PROGRAM TempCtrl
VAR

END_VAR

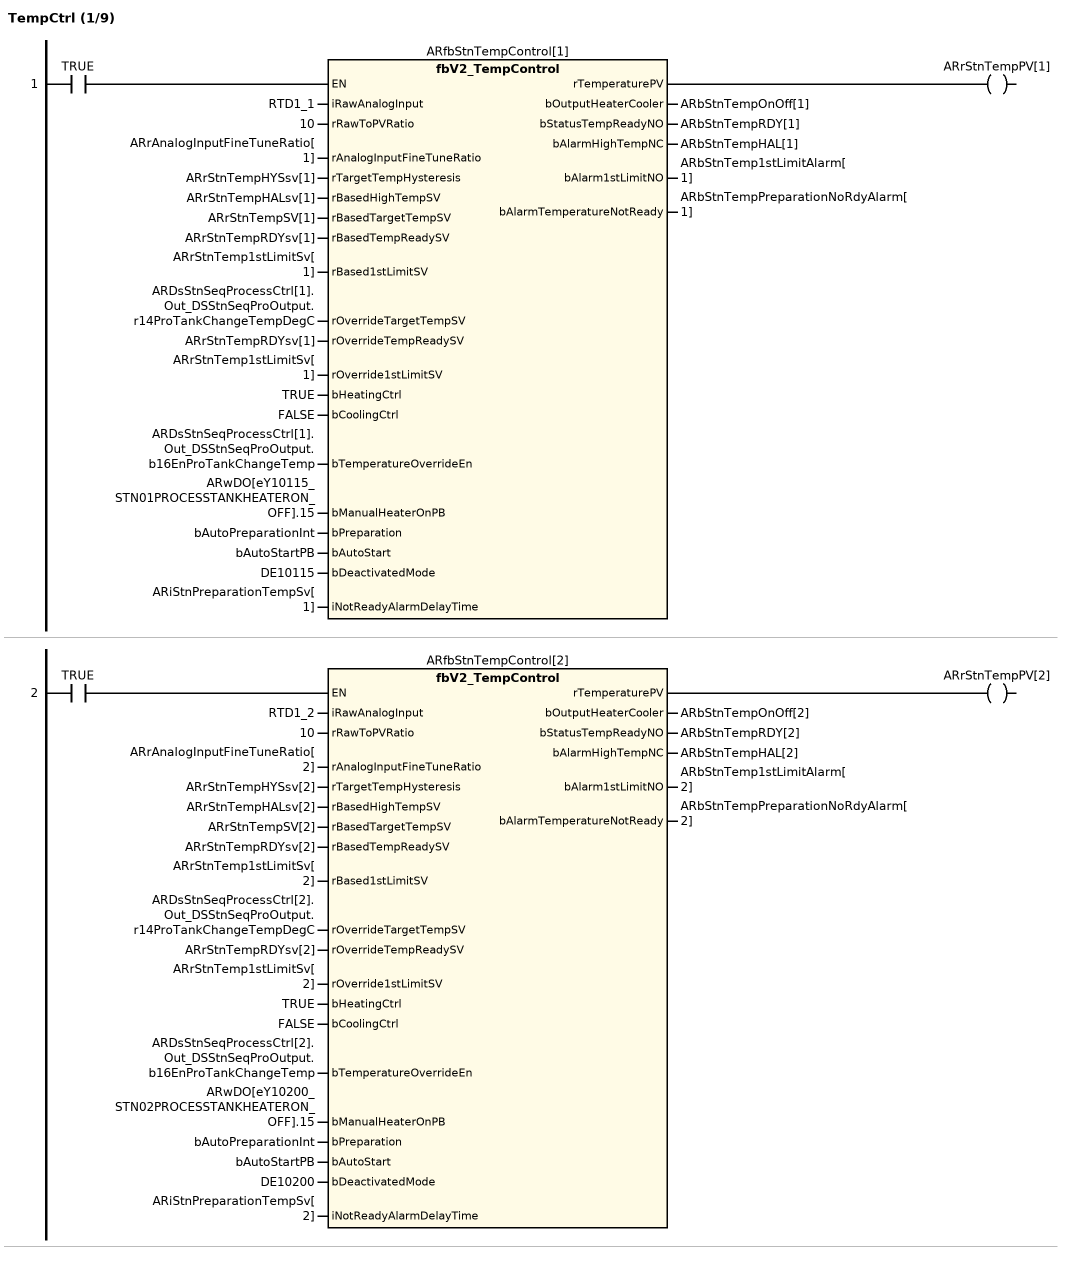
// NETWORK 1
ARfbStnTempControl[1](
    iRawAnalogInput := RTD1_1,
    rRawToPVRatio := 10,
    rAnalogInputFineTuneRatio := ARrAnalogInputFineTuneRatio[1],
    rTargetTempHysteresis := ARrStnTempHYSsv[1],
    rBasedHighTempSV := ARrStnTempHALsv[1],
    rBasedTargetTempSV := ARrStnTempSV[1],
    rBasedTempReadySV := ARrStnTempRDYsv[1],
    rBased1stLimitSV := ARrStnTemp1stLimitSv[1],
    rOverrideTargetTempSV := ARDsStnSeqProcessCtrl[1].Out_DSStnSeqProOutput.r14ProTankChangeTempDegC,
    rOverrideTempReadySV := ARrStnTempRDYsv[1],
    rOverride1stLimitSV := ARrStnTemp1stLimitSv[1],
    bHeatingCtrl := TRUE,
    bCoolingCtrl := FALSE,
    bTemperatureOverrideEn := ARDsStnSeqProcessCtrl[1].Out_DSStnSeqProOutput.b16EnProTankChangeTemp,
    bManualHeaterOnPB := ARwDO[eY10115_STN01PROCESSTANKHEATERON_OFF].15,
    bPreparation := bAutoPreparationInt,
    bAutoStart := bAutoStartPB,
    bDeactivatedMode := DE10115,
    iNotReadyAlarmDelayTime := ARiStnPreparationTempSv[1],
    bOutputHeaterCooler => ARbStnTempOnOff[1],
    bStatusTempReadyNO => ARbStnTempRDY[1],
    bAlarmHighTempNC => ARbStnTempHAL[1],
    bAlarm1stLimitNO => ARbStnTemp1stLimitAlarm[1],
    bAlarmTemperatureNotReady => ARbStnTempPreparationNoRdyAlarm[1]); // fbV2_TempControl
ARrStnTempPV[1] := ARfbStnTempControl[1].rTemperaturePV;

// NETWORK 2
ARfbStnTempControl[2](
    iRawAnalogInput := RTD1_2,
    rRawToPVRatio := 10,
    rAnalogInputFineTuneRatio := ARrAnalogInputFineTuneRatio[2],
    rTargetTempHysteresis := ARrStnTempHYSsv[2],
    rBasedHighTempSV := ARrStnTempHALsv[2],
    rBasedTargetTempSV := ARrStnTempSV[2],
    rBasedTempReadySV := ARrStnTempRDYsv[2],
    rBased1stLimitSV := ARrStnTemp1stLimitSv[2],
    rOverrideTargetTempSV := ARDsStnSeqProcessCtrl[2].Out_DSStnSeqProOutput.r14ProTankChangeTempDegC,
    rOverrideTempReadySV := ARrStnTempRDYsv[2],
    rOverride1stLimitSV := ARrStnTemp1stLimitSv[2],
    bHeatingCtrl := TRUE,
    bCoolingCtrl := FALSE,
    bTemperatureOverrideEn := ARDsStnSeqProcessCtrl[2].Out_DSStnSeqProOutput.b16EnProTankChangeTemp,
    bManualHeaterOnPB := ARwDO[eY10200_STN02PROCESSTANKHEATERON_OFF].15,
    bPreparation := bAutoPreparationInt,
    bAutoStart := bAutoStartPB,
    bDeactivatedMode := DE10200,
    iNotReadyAlarmDelayTime := ARiStnPreparationTempSv[2],
    bOutputHeaterCooler => ARbStnTempOnOff[2],
    bStatusTempReadyNO => ARbStnTempRDY[2],
    bAlarmHighTempNC => ARbStnTempHAL[2],
    bAlarm1stLimitNO => ARbStnTemp1stLimitAlarm[2],
    bAlarmTemperatureNotReady => ARbStnTempPreparationNoRdyAlarm[2]); // fbV2_TempControl
ARrStnTempPV[2] := ARfbStnTempControl[2].rTemperaturePV;

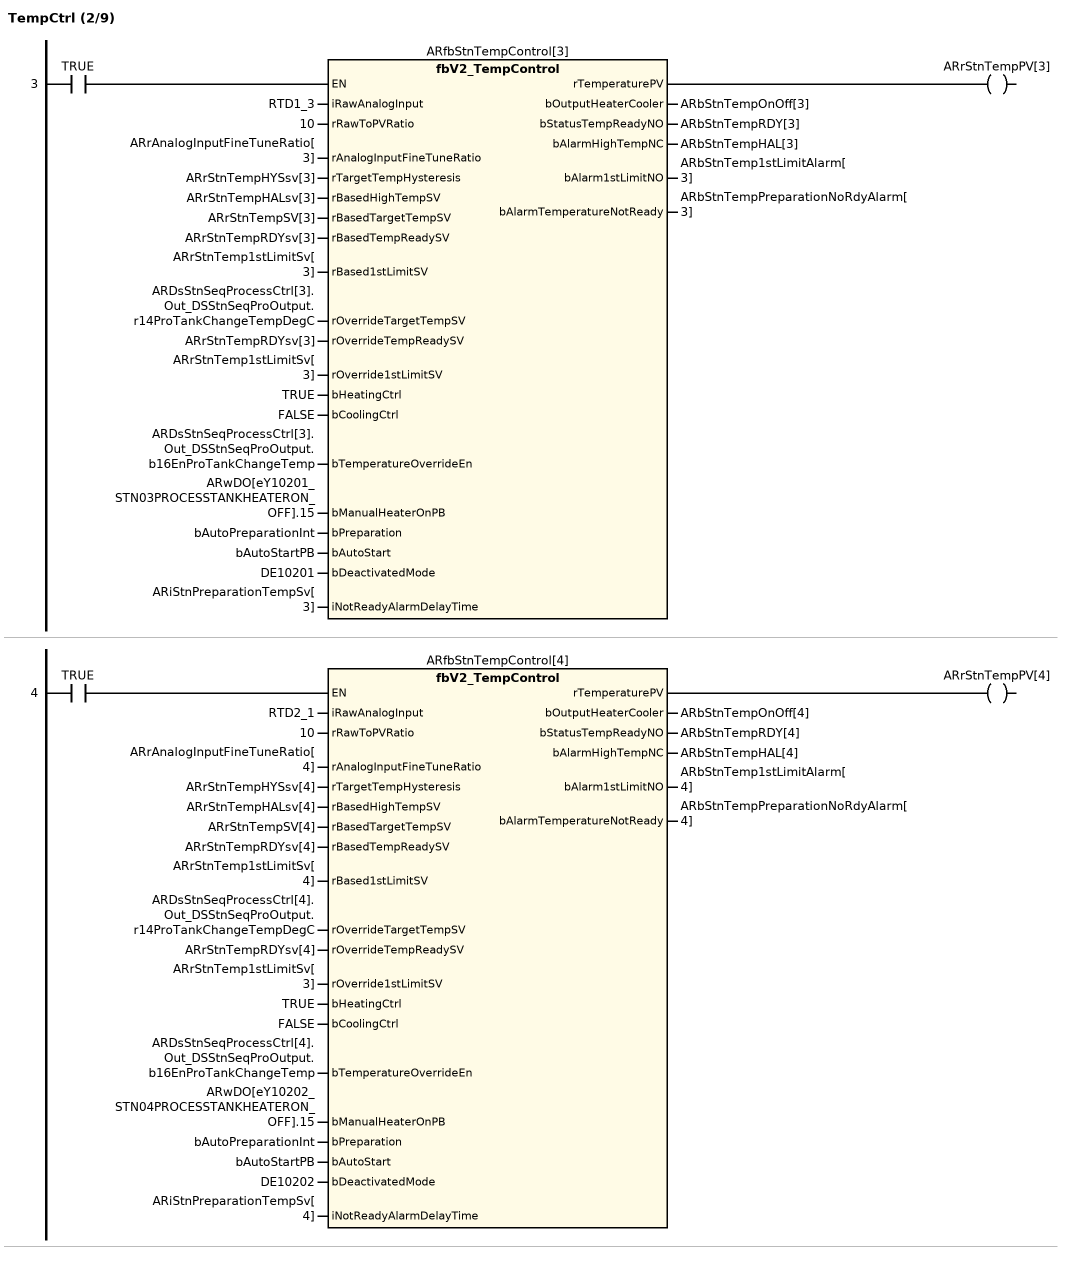
// NETWORK 3
ARfbStnTempControl[3](
    iRawAnalogInput := RTD1_3,
    rRawToPVRatio := 10,
    rAnalogInputFineTuneRatio := ARrAnalogInputFineTuneRatio[3],
    rTargetTempHysteresis := ARrStnTempHYSsv[3],
    rBasedHighTempSV := ARrStnTempHALsv[3],
    rBasedTargetTempSV := ARrStnTempSV[3],
    rBasedTempReadySV := ARrStnTempRDYsv[3],
    rBased1stLimitSV := ARrStnTemp1stLimitSv[3],
    rOverrideTargetTempSV := ARDsStnSeqProcessCtrl[3].Out_DSStnSeqProOutput.r14ProTankChangeTempDegC,
    rOverrideTempReadySV := ARrStnTempRDYsv[3],
    rOverride1stLimitSV := ARrStnTemp1stLimitSv[3],
    bHeatingCtrl := TRUE,
    bCoolingCtrl := FALSE,
    bTemperatureOverrideEn := ARDsStnSeqProcessCtrl[3].Out_DSStnSeqProOutput.b16EnProTankChangeTemp,
    bManualHeaterOnPB := ARwDO[eY10201_STN03PROCESSTANKHEATERON_OFF].15,
    bPreparation := bAutoPreparationInt,
    bAutoStart := bAutoStartPB,
    bDeactivatedMode := DE10201,
    iNotReadyAlarmDelayTime := ARiStnPreparationTempSv[3],
    bOutputHeaterCooler => ARbStnTempOnOff[3],
    bStatusTempReadyNO => ARbStnTempRDY[3],
    bAlarmHighTempNC => ARbStnTempHAL[3],
    bAlarm1stLimitNO => ARbStnTemp1stLimitAlarm[3],
    bAlarmTemperatureNotReady => ARbStnTempPreparationNoRdyAlarm[3]); // fbV2_TempControl
ARrStnTempPV[3] := ARfbStnTempControl[3].rTemperaturePV;

// NETWORK 4
ARfbStnTempControl[4](
    iRawAnalogInput := RTD2_1,
    rRawToPVRatio := 10,
    rAnalogInputFineTuneRatio := ARrAnalogInputFineTuneRatio[4],
    rTargetTempHysteresis := ARrStnTempHYSsv[4],
    rBasedHighTempSV := ARrStnTempHALsv[4],
    rBasedTargetTempSV := ARrStnTempSV[4],
    rBasedTempReadySV := ARrStnTempRDYsv[4],
    rBased1stLimitSV := ARrStnTemp1stLimitSv[4],
    rOverrideTargetTempSV := ARDsStnSeqProcessCtrl[4].Out_DSStnSeqProOutput.r14ProTankChangeTempDegC,
    rOverrideTempReadySV := ARrStnTempRDYsv[4],
    rOverride1stLimitSV := ARrStnTemp1stLimitSv[3],
    bHeatingCtrl := TRUE,
    bCoolingCtrl := FALSE,
    bTemperatureOverrideEn := ARDsStnSeqProcessCtrl[4].Out_DSStnSeqProOutput.b16EnProTankChangeTemp,
    bManualHeaterOnPB := ARwDO[eY10202_STN04PROCESSTANKHEATERON_OFF].15,
    bPreparation := bAutoPreparationInt,
    bAutoStart := bAutoStartPB,
    bDeactivatedMode := DE10202,
    iNotReadyAlarmDelayTime := ARiStnPreparationTempSv[4],
    bOutputHeaterCooler => ARbStnTempOnOff[4],
    bStatusTempReadyNO => ARbStnTempRDY[4],
    bAlarmHighTempNC => ARbStnTempHAL[4],
    bAlarm1stLimitNO => ARbStnTemp1stLimitAlarm[4],
    bAlarmTemperatureNotReady => ARbStnTempPreparationNoRdyAlarm[4]); // fbV2_TempControl
ARrStnTempPV[4] := ARfbStnTempControl[4].rTemperaturePV;

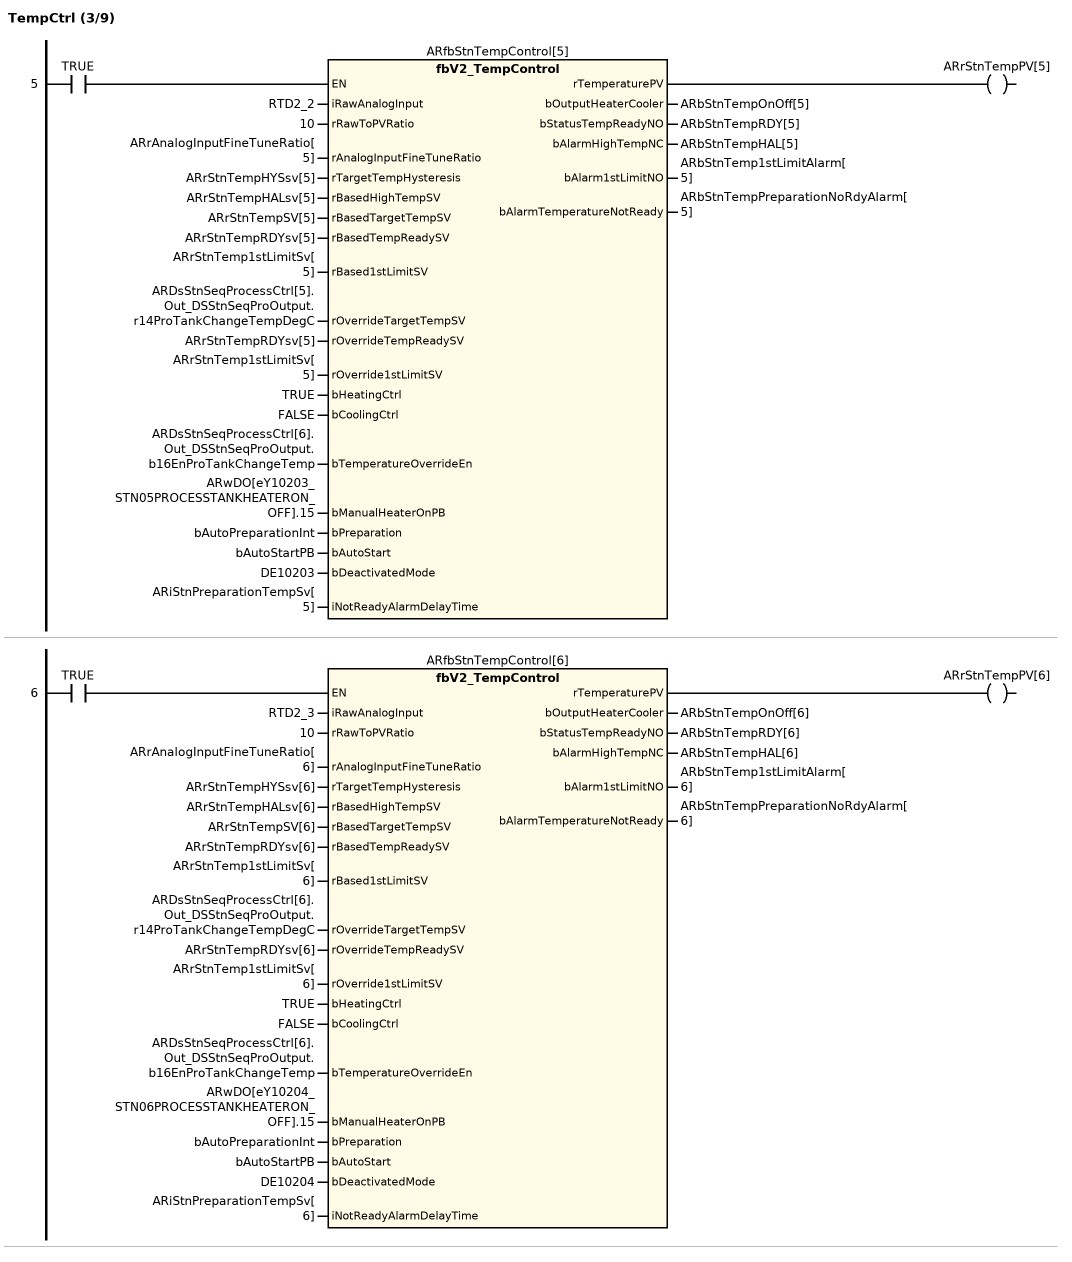
// NETWORK 5
ARfbStnTempControl[5](
    iRawAnalogInput := RTD2_2,
    rRawToPVRatio := 10,
    rAnalogInputFineTuneRatio := ARrAnalogInputFineTuneRatio[5],
    rTargetTempHysteresis := ARrStnTempHYSsv[5],
    rBasedHighTempSV := ARrStnTempHALsv[5],
    rBasedTargetTempSV := ARrStnTempSV[5],
    rBasedTempReadySV := ARrStnTempRDYsv[5],
    rBased1stLimitSV := ARrStnTemp1stLimitSv[5],
    rOverrideTargetTempSV := ARDsStnSeqProcessCtrl[5].Out_DSStnSeqProOutput.r14ProTankChangeTempDegC,
    rOverrideTempReadySV := ARrStnTempRDYsv[5],
    rOverride1stLimitSV := ARrStnTemp1stLimitSv[5],
    bHeatingCtrl := TRUE,
    bCoolingCtrl := FALSE,
    bTemperatureOverrideEn := ARDsStnSeqProcessCtrl[6].Out_DSStnSeqProOutput.b16EnProTankChangeTemp,
    bManualHeaterOnPB := ARwDO[eY10203_STN05PROCESSTANKHEATERON_OFF].15,
    bPreparation := bAutoPreparationInt,
    bAutoStart := bAutoStartPB,
    bDeactivatedMode := DE10203,
    iNotReadyAlarmDelayTime := ARiStnPreparationTempSv[5],
    bOutputHeaterCooler => ARbStnTempOnOff[5],
    bStatusTempReadyNO => ARbStnTempRDY[5],
    bAlarmHighTempNC => ARbStnTempHAL[5],
    bAlarm1stLimitNO => ARbStnTemp1stLimitAlarm[5],
    bAlarmTemperatureNotReady => ARbStnTempPreparationNoRdyAlarm[5]); // fbV2_TempControl
ARrStnTempPV[5] := ARfbStnTempControl[5].rTemperaturePV;

// NETWORK 6
ARfbStnTempControl[6](
    iRawAnalogInput := RTD2_3,
    rRawToPVRatio := 10,
    rAnalogInputFineTuneRatio := ARrAnalogInputFineTuneRatio[6],
    rTargetTempHysteresis := ARrStnTempHYSsv[6],
    rBasedHighTempSV := ARrStnTempHALsv[6],
    rBasedTargetTempSV := ARrStnTempSV[6],
    rBasedTempReadySV := ARrStnTempRDYsv[6],
    rBased1stLimitSV := ARrStnTemp1stLimitSv[6],
    rOverrideTargetTempSV := ARDsStnSeqProcessCtrl[6].Out_DSStnSeqProOutput.r14ProTankChangeTempDegC,
    rOverrideTempReadySV := ARrStnTempRDYsv[6],
    rOverride1stLimitSV := ARrStnTemp1stLimitSv[6],
    bHeatingCtrl := TRUE,
    bCoolingCtrl := FALSE,
    bTemperatureOverrideEn := ARDsStnSeqProcessCtrl[6].Out_DSStnSeqProOutput.b16EnProTankChangeTemp,
    bManualHeaterOnPB := ARwDO[eY10204_STN06PROCESSTANKHEATERON_OFF].15,
    bPreparation := bAutoPreparationInt,
    bAutoStart := bAutoStartPB,
    bDeactivatedMode := DE10204,
    iNotReadyAlarmDelayTime := ARiStnPreparationTempSv[6],
    bOutputHeaterCooler => ARbStnTempOnOff[6],
    bStatusTempReadyNO => ARbStnTempRDY[6],
    bAlarmHighTempNC => ARbStnTempHAL[6],
    bAlarm1stLimitNO => ARbStnTemp1stLimitAlarm[6],
    bAlarmTemperatureNotReady => ARbStnTempPreparationNoRdyAlarm[6]); // fbV2_TempControl
ARrStnTempPV[6] := ARfbStnTempControl[6].rTemperaturePV;

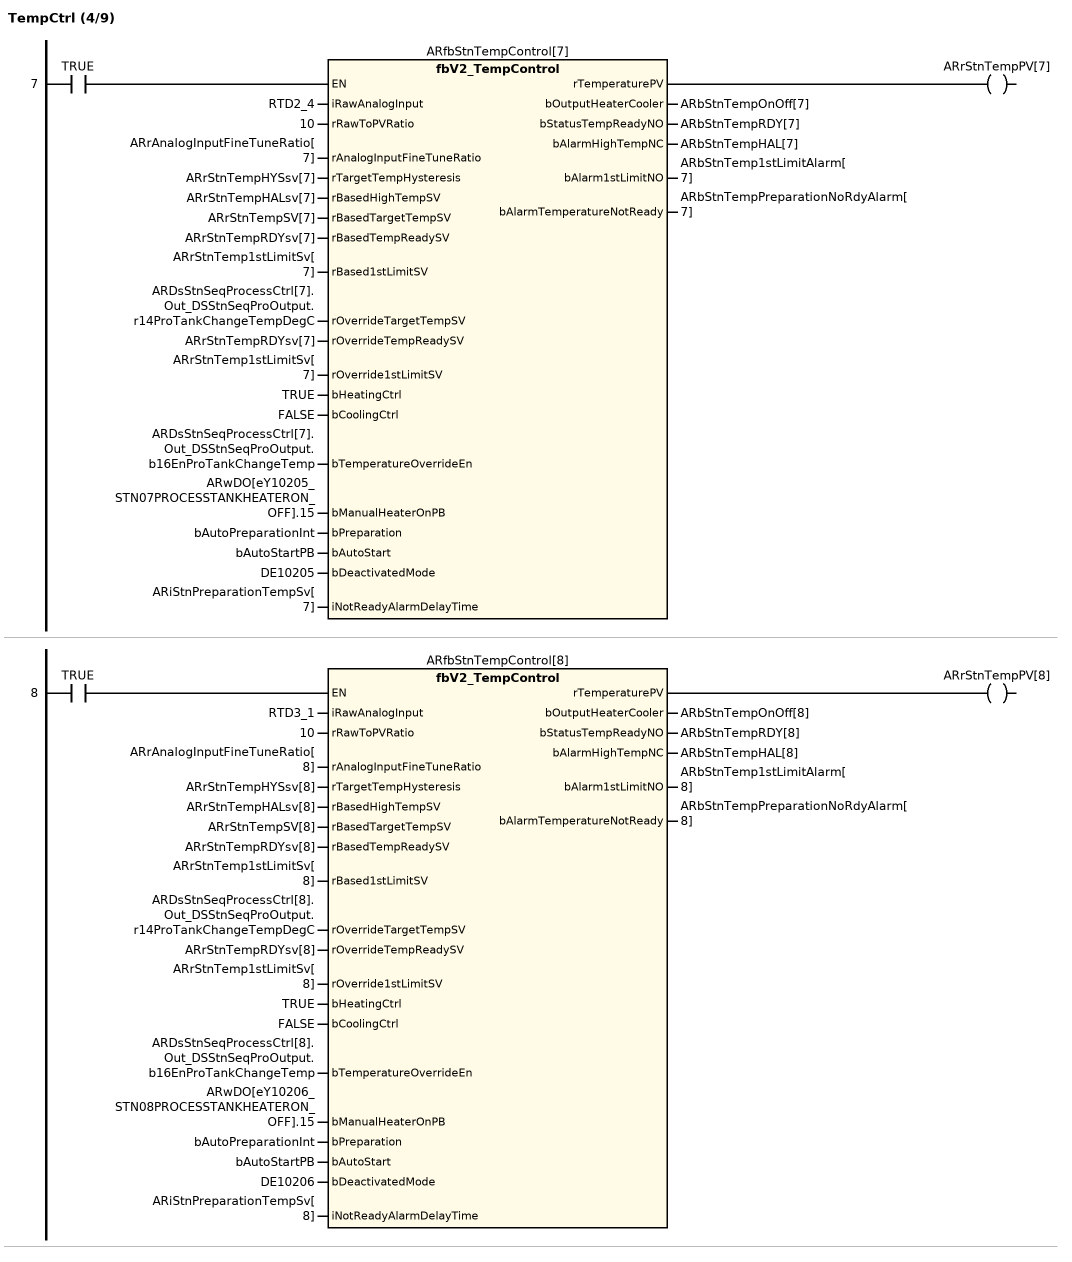
// NETWORK 7
ARfbStnTempControl[7](
    iRawAnalogInput := RTD2_4,
    rRawToPVRatio := 10,
    rAnalogInputFineTuneRatio := ARrAnalogInputFineTuneRatio[7],
    rTargetTempHysteresis := ARrStnTempHYSsv[7],
    rBasedHighTempSV := ARrStnTempHALsv[7],
    rBasedTargetTempSV := ARrStnTempSV[7],
    rBasedTempReadySV := ARrStnTempRDYsv[7],
    rBased1stLimitSV := ARrStnTemp1stLimitSv[7],
    rOverrideTargetTempSV := ARDsStnSeqProcessCtrl[7].Out_DSStnSeqProOutput.r14ProTankChangeTempDegC,
    rOverrideTempReadySV := ARrStnTempRDYsv[7],
    rOverride1stLimitSV := ARrStnTemp1stLimitSv[7],
    bHeatingCtrl := TRUE,
    bCoolingCtrl := FALSE,
    bTemperatureOverrideEn := ARDsStnSeqProcessCtrl[7].Out_DSStnSeqProOutput.b16EnProTankChangeTemp,
    bManualHeaterOnPB := ARwDO[eY10205_STN07PROCESSTANKHEATERON_OFF].15,
    bPreparation := bAutoPreparationInt,
    bAutoStart := bAutoStartPB,
    bDeactivatedMode := DE10205,
    iNotReadyAlarmDelayTime := ARiStnPreparationTempSv[7],
    bOutputHeaterCooler => ARbStnTempOnOff[7],
    bStatusTempReadyNO => ARbStnTempRDY[7],
    bAlarmHighTempNC => ARbStnTempHAL[7],
    bAlarm1stLimitNO => ARbStnTemp1stLimitAlarm[7],
    bAlarmTemperatureNotReady => ARbStnTempPreparationNoRdyAlarm[7]); // fbV2_TempControl
ARrStnTempPV[7] := ARfbStnTempControl[7].rTemperaturePV;

// NETWORK 8
ARfbStnTempControl[8](
    iRawAnalogInput := RTD3_1,
    rRawToPVRatio := 10,
    rAnalogInputFineTuneRatio := ARrAnalogInputFineTuneRatio[8],
    rTargetTempHysteresis := ARrStnTempHYSsv[8],
    rBasedHighTempSV := ARrStnTempHALsv[8],
    rBasedTargetTempSV := ARrStnTempSV[8],
    rBasedTempReadySV := ARrStnTempRDYsv[8],
    rBased1stLimitSV := ARrStnTemp1stLimitSv[8],
    rOverrideTargetTempSV := ARDsStnSeqProcessCtrl[8].Out_DSStnSeqProOutput.r14ProTankChangeTempDegC,
    rOverrideTempReadySV := ARrStnTempRDYsv[8],
    rOverride1stLimitSV := ARrStnTemp1stLimitSv[8],
    bHeatingCtrl := TRUE,
    bCoolingCtrl := FALSE,
    bTemperatureOverrideEn := ARDsStnSeqProcessCtrl[8].Out_DSStnSeqProOutput.b16EnProTankChangeTemp,
    bManualHeaterOnPB := ARwDO[eY10206_STN08PROCESSTANKHEATERON_OFF].15,
    bPreparation := bAutoPreparationInt,
    bAutoStart := bAutoStartPB,
    bDeactivatedMode := DE10206,
    iNotReadyAlarmDelayTime := ARiStnPreparationTempSv[8],
    bOutputHeaterCooler => ARbStnTempOnOff[8],
    bStatusTempReadyNO => ARbStnTempRDY[8],
    bAlarmHighTempNC => ARbStnTempHAL[8],
    bAlarm1stLimitNO => ARbStnTemp1stLimitAlarm[8],
    bAlarmTemperatureNotReady => ARbStnTempPreparationNoRdyAlarm[8]); // fbV2_TempControl
ARrStnTempPV[8] := ARfbStnTempControl[8].rTemperaturePV;

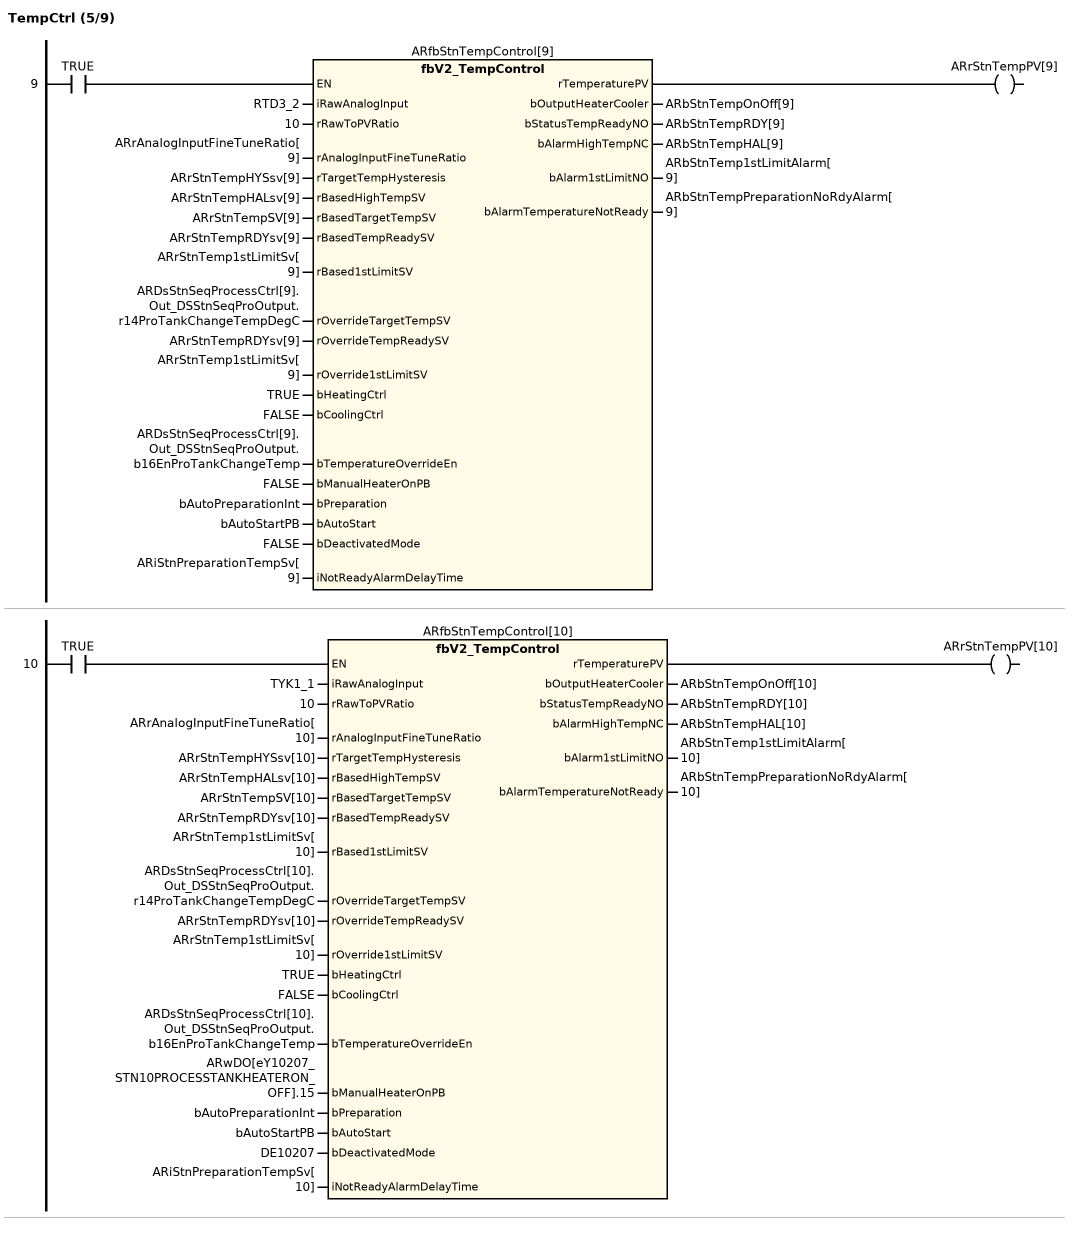
// NETWORK 9
ARfbStnTempControl[9](
    iRawAnalogInput := RTD3_2,
    rRawToPVRatio := 10,
    rAnalogInputFineTuneRatio := ARrAnalogInputFineTuneRatio[9],
    rTargetTempHysteresis := ARrStnTempHYSsv[9],
    rBasedHighTempSV := ARrStnTempHALsv[9],
    rBasedTargetTempSV := ARrStnTempSV[9],
    rBasedTempReadySV := ARrStnTempRDYsv[9],
    rBased1stLimitSV := ARrStnTemp1stLimitSv[9],
    rOverrideTargetTempSV := ARDsStnSeqProcessCtrl[9].Out_DSStnSeqProOutput.r14ProTankChangeTempDegC,
    rOverrideTempReadySV := ARrStnTempRDYsv[9],
    rOverride1stLimitSV := ARrStnTemp1stLimitSv[9],
    bHeatingCtrl := TRUE,
    bCoolingCtrl := FALSE,
    bTemperatureOverrideEn := ARDsStnSeqProcessCtrl[9].Out_DSStnSeqProOutput.b16EnProTankChangeTemp,
    bManualHeaterOnPB := FALSE,
    bPreparation := bAutoPreparationInt,
    bAutoStart := bAutoStartPB,
    bDeactivatedMode := FALSE,
    iNotReadyAlarmDelayTime := ARiStnPreparationTempSv[9],
    bOutputHeaterCooler => ARbStnTempOnOff[9],
    bStatusTempReadyNO => ARbStnTempRDY[9],
    bAlarmHighTempNC => ARbStnTempHAL[9],
    bAlarm1stLimitNO => ARbStnTemp1stLimitAlarm[9],
    bAlarmTemperatureNotReady => ARbStnTempPreparationNoRdyAlarm[9]); // fbV2_TempControl
ARrStnTempPV[9] := ARfbStnTempControl[9].rTemperaturePV;

// NETWORK 10
ARfbStnTempControl[10](
    iRawAnalogInput := TYK1_1,
    rRawToPVRatio := 10,
    rAnalogInputFineTuneRatio := ARrAnalogInputFineTuneRatio[10],
    rTargetTempHysteresis := ARrStnTempHYSsv[10],
    rBasedHighTempSV := ARrStnTempHALsv[10],
    rBasedTargetTempSV := ARrStnTempSV[10],
    rBasedTempReadySV := ARrStnTempRDYsv[10],
    rBased1stLimitSV := ARrStnTemp1stLimitSv[10],
    rOverrideTargetTempSV := ARDsStnSeqProcessCtrl[10].Out_DSStnSeqProOutput.r14ProTankChangeTempDegC,
    rOverrideTempReadySV := ARrStnTempRDYsv[10],
    rOverride1stLimitSV := ARrStnTemp1stLimitSv[10],
    bHeatingCtrl := TRUE,
    bCoolingCtrl := FALSE,
    bTemperatureOverrideEn := ARDsStnSeqProcessCtrl[10].Out_DSStnSeqProOutput.b16EnProTankChangeTemp,
    bManualHeaterOnPB := ARwDO[eY10207_STN10PROCESSTANKHEATERON_OFF].15,
    bPreparation := bAutoPreparationInt,
    bAutoStart := bAutoStartPB,
    bDeactivatedMode := DE10207,
    iNotReadyAlarmDelayTime := ARiStnPreparationTempSv[10],
    bOutputHeaterCooler => ARbStnTempOnOff[10],
    bStatusTempReadyNO => ARbStnTempRDY[10],
    bAlarmHighTempNC => ARbStnTempHAL[10],
    bAlarm1stLimitNO => ARbStnTemp1stLimitAlarm[10],
    bAlarmTemperatureNotReady => ARbStnTempPreparationNoRdyAlarm[10]); // fbV2_TempControl
ARrStnTempPV[10] := ARfbStnTempControl[10].rTemperaturePV;

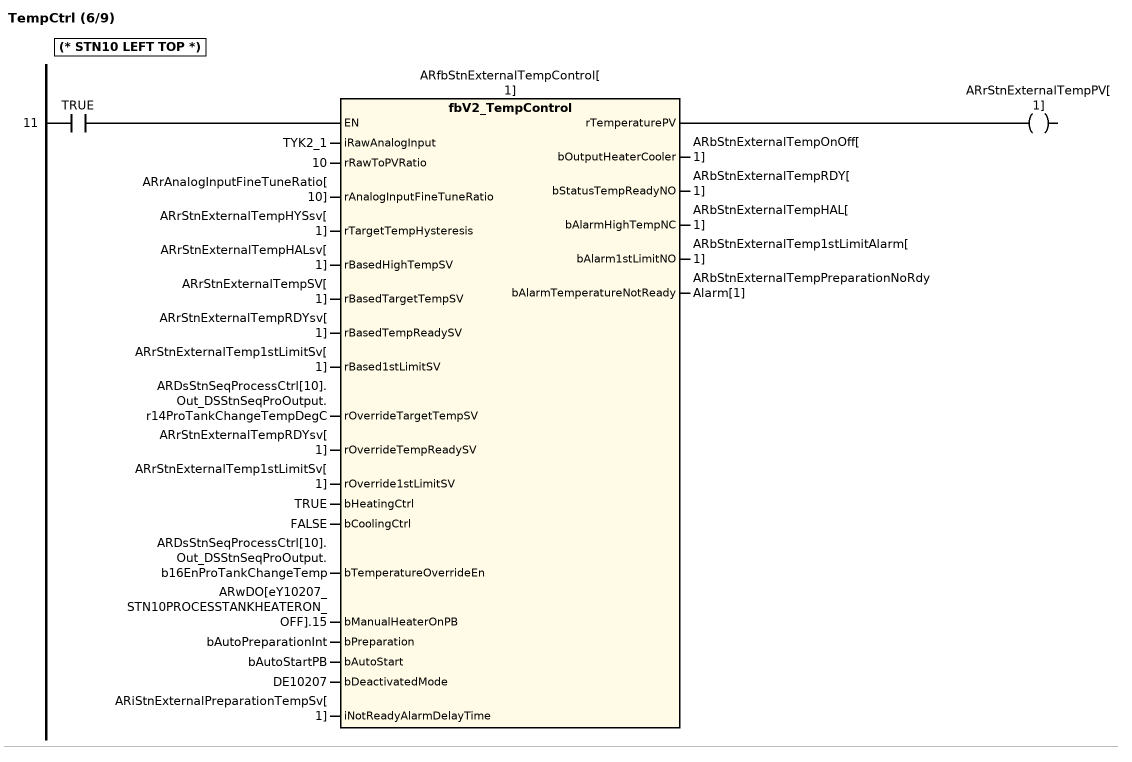
// NETWORK 11
// label: (* STN10 LEFT TOP *)
ARfbStnExternalTempControl[1](
    iRawAnalogInput := TYK2_1,
    rRawToPVRatio := 10,
    rAnalogInputFineTuneRatio := ARrAnalogInputFineTuneRatio[10],
    rTargetTempHysteresis := ARrStnExternalTempHYSsv[1],
    rBasedHighTempSV := ARrStnExternalTempHALsv[1],
    rBasedTargetTempSV := ARrStnExternalTempSV[1],
    rBasedTempReadySV := ARrStnExternalTempRDYsv[1],
    rBased1stLimitSV := ARrStnExternalTemp1stLimitSv[1],
    rOverrideTargetTempSV := ARDsStnSeqProcessCtrl[10].Out_DSStnSeqProOutput.r14ProTankChangeTempDegC,
    rOverrideTempReadySV := ARrStnExternalTempRDYsv[1],
    rOverride1stLimitSV := ARrStnExternalTemp1stLimitSv[1],
    bHeatingCtrl := TRUE,
    bCoolingCtrl := FALSE,
    bTemperatureOverrideEn := ARDsStnSeqProcessCtrl[10].Out_DSStnSeqProOutput.b16EnProTankChangeTemp,
    bManualHeaterOnPB := ARwDO[eY10207_STN10PROCESSTANKHEATERON_OFF].15,
    bPreparation := bAutoPreparationInt,
    bAutoStart := bAutoStartPB,
    bDeactivatedMode := DE10207,
    iNotReadyAlarmDelayTime := ARiStnExternalPreparationTempSv[1],
    bOutputHeaterCooler => ARbStnExternalTempOnOff[1],
    bStatusTempReadyNO => ARbStnExternalTempRDY[1],
    bAlarmHighTempNC => ARbStnExternalTempHAL[1],
    bAlarm1stLimitNO => ARbStnExternalTemp1stLimitAlarm[1],
    bAlarmTemperatureNotReady => ARbStnExternalTempPreparationNoRdyAlarm[1]); // fbV2_TempControl
ARrStnExternalTempPV[1] := ARfbStnExternalTempControl[1].rTemperaturePV;

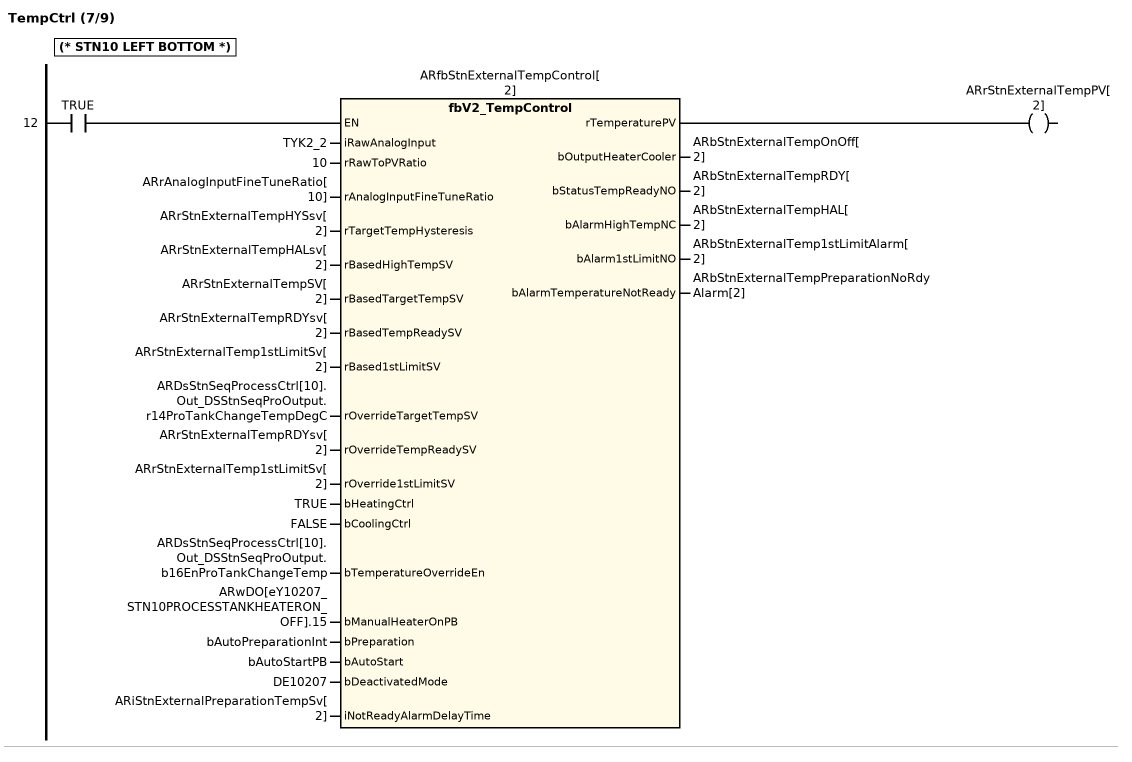
// NETWORK 12
// label: (* STN10 LEFT BOTTOM *)
ARfbStnExternalTempControl[2](
    iRawAnalogInput := TYK2_2,
    rRawToPVRatio := 10,
    rAnalogInputFineTuneRatio := ARrAnalogInputFineTuneRatio[10],
    rTargetTempHysteresis := ARrStnExternalTempHYSsv[2],
    rBasedHighTempSV := ARrStnExternalTempHALsv[2],
    rBasedTargetTempSV := ARrStnExternalTempSV[2],
    rBasedTempReadySV := ARrStnExternalTempRDYsv[2],
    rBased1stLimitSV := ARrStnExternalTemp1stLimitSv[2],
    rOverrideTargetTempSV := ARDsStnSeqProcessCtrl[10].Out_DSStnSeqProOutput.r14ProTankChangeTempDegC,
    rOverrideTempReadySV := ARrStnExternalTempRDYsv[2],
    rOverride1stLimitSV := ARrStnExternalTemp1stLimitSv[2],
    bHeatingCtrl := TRUE,
    bCoolingCtrl := FALSE,
    bTemperatureOverrideEn := ARDsStnSeqProcessCtrl[10].Out_DSStnSeqProOutput.b16EnProTankChangeTemp,
    bManualHeaterOnPB := ARwDO[eY10207_STN10PROCESSTANKHEATERON_OFF].15,
    bPreparation := bAutoPreparationInt,
    bAutoStart := bAutoStartPB,
    bDeactivatedMode := DE10207,
    iNotReadyAlarmDelayTime := ARiStnExternalPreparationTempSv[2],
    bOutputHeaterCooler => ARbStnExternalTempOnOff[2],
    bStatusTempReadyNO => ARbStnExternalTempRDY[2],
    bAlarmHighTempNC => ARbStnExternalTempHAL[2],
    bAlarm1stLimitNO => ARbStnExternalTemp1stLimitAlarm[2],
    bAlarmTemperatureNotReady => ARbStnExternalTempPreparationNoRdyAlarm[2]); // fbV2_TempControl
ARrStnExternalTempPV[2] := ARfbStnExternalTempControl[2].rTemperaturePV;

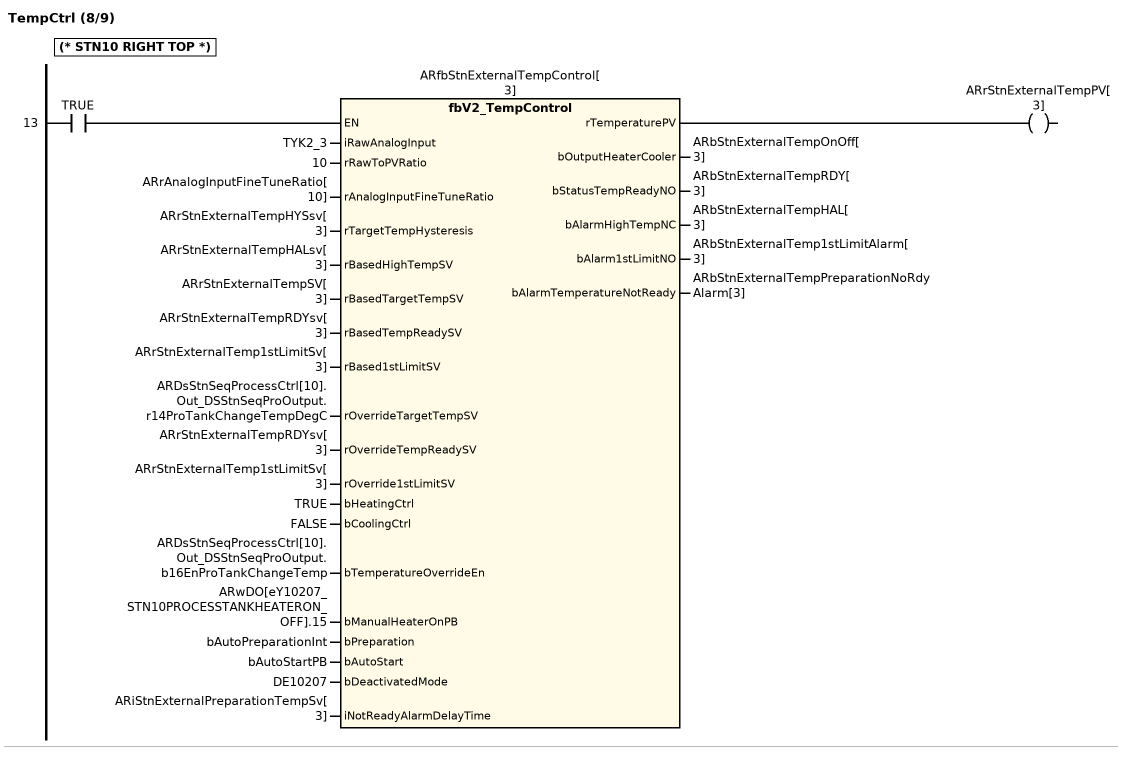
// NETWORK 13
// label: (* STN10 RIGHT TOP *)
ARfbStnExternalTempControl[3](
    iRawAnalogInput := TYK2_3,
    rRawToPVRatio := 10,
    rAnalogInputFineTuneRatio := ARrAnalogInputFineTuneRatio[10],
    rTargetTempHysteresis := ARrStnExternalTempHYSsv[3],
    rBasedHighTempSV := ARrStnExternalTempHALsv[3],
    rBasedTargetTempSV := ARrStnExternalTempSV[3],
    rBasedTempReadySV := ARrStnExternalTempRDYsv[3],
    rBased1stLimitSV := ARrStnExternalTemp1stLimitSv[3],
    rOverrideTargetTempSV := ARDsStnSeqProcessCtrl[10].Out_DSStnSeqProOutput.r14ProTankChangeTempDegC,
    rOverrideTempReadySV := ARrStnExternalTempRDYsv[3],
    rOverride1stLimitSV := ARrStnExternalTemp1stLimitSv[3],
    bHeatingCtrl := TRUE,
    bCoolingCtrl := FALSE,
    bTemperatureOverrideEn := ARDsStnSeqProcessCtrl[10].Out_DSStnSeqProOutput.b16EnProTankChangeTemp,
    bManualHeaterOnPB := ARwDO[eY10207_STN10PROCESSTANKHEATERON_OFF].15,
    bPreparation := bAutoPreparationInt,
    bAutoStart := bAutoStartPB,
    bDeactivatedMode := DE10207,
    iNotReadyAlarmDelayTime := ARiStnExternalPreparationTempSv[3],
    bOutputHeaterCooler => ARbStnExternalTempOnOff[3],
    bStatusTempReadyNO => ARbStnExternalTempRDY[3],
    bAlarmHighTempNC => ARbStnExternalTempHAL[3],
    bAlarm1stLimitNO => ARbStnExternalTemp1stLimitAlarm[3],
    bAlarmTemperatureNotReady => ARbStnExternalTempPreparationNoRdyAlarm[3]); // fbV2_TempControl
ARrStnExternalTempPV[3] := ARfbStnExternalTempControl[3].rTemperaturePV;

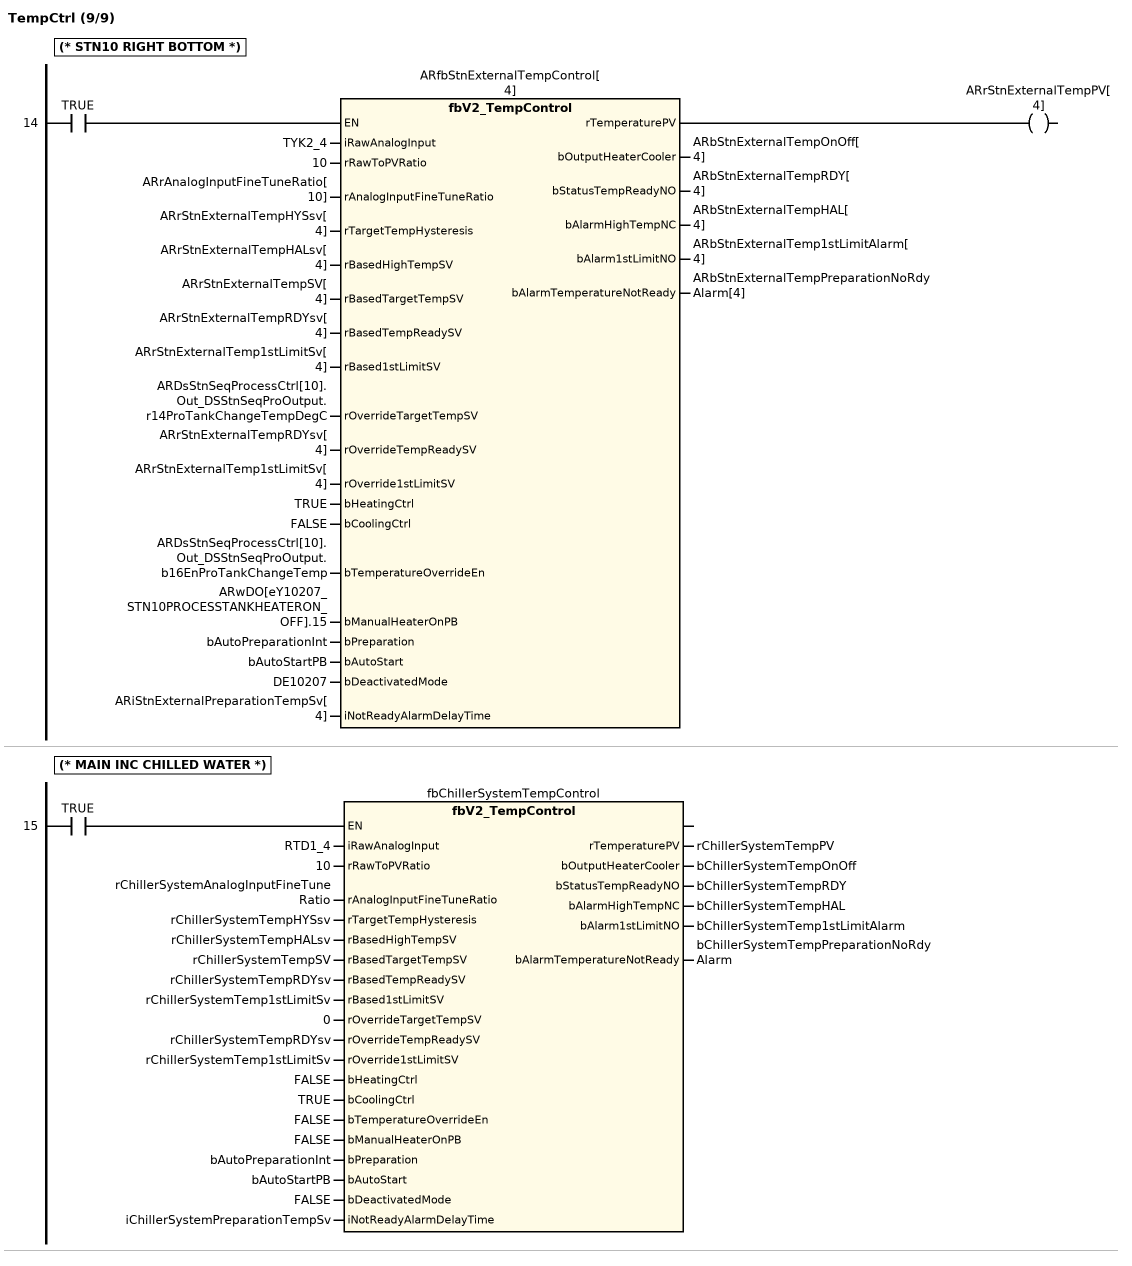
// NETWORK 14
// label: (* STN10 RIGHT BOTTOM *)
ARfbStnExternalTempControl[4](
    iRawAnalogInput := TYK2_4,
    rRawToPVRatio := 10,
    rAnalogInputFineTuneRatio := ARrAnalogInputFineTuneRatio[10],
    rTargetTempHysteresis := ARrStnExternalTempHYSsv[4],
    rBasedHighTempSV := ARrStnExternalTempHALsv[4],
    rBasedTargetTempSV := ARrStnExternalTempSV[4],
    rBasedTempReadySV := ARrStnExternalTempRDYsv[4],
    rBased1stLimitSV := ARrStnExternalTemp1stLimitSv[4],
    rOverrideTargetTempSV := ARDsStnSeqProcessCtrl[10].Out_DSStnSeqProOutput.r14ProTankChangeTempDegC,
    rOverrideTempReadySV := ARrStnExternalTempRDYsv[4],
    rOverride1stLimitSV := ARrStnExternalTemp1stLimitSv[4],
    bHeatingCtrl := TRUE,
    bCoolingCtrl := FALSE,
    bTemperatureOverrideEn := ARDsStnSeqProcessCtrl[10].Out_DSStnSeqProOutput.b16EnProTankChangeTemp,
    bManualHeaterOnPB := ARwDO[eY10207_STN10PROCESSTANKHEATERON_OFF].15,
    bPreparation := bAutoPreparationInt,
    bAutoStart := bAutoStartPB,
    bDeactivatedMode := DE10207,
    iNotReadyAlarmDelayTime := ARiStnExternalPreparationTempSv[4],
    bOutputHeaterCooler => ARbStnExternalTempOnOff[4],
    bStatusTempReadyNO => ARbStnExternalTempRDY[4],
    bAlarmHighTempNC => ARbStnExternalTempHAL[4],
    bAlarm1stLimitNO => ARbStnExternalTemp1stLimitAlarm[4],
    bAlarmTemperatureNotReady => ARbStnExternalTempPreparationNoRdyAlarm[4]); // fbV2_TempControl
ARrStnExternalTempPV[4] := ARfbStnExternalTempControl[4].rTemperaturePV;

// NETWORK 15
// label: (* MAIN INC CHILLED WATER *)
fbChillerSystemTempControl(
    iRawAnalogInput := RTD1_4,
    rRawToPVRatio := 10,
    rAnalogInputFineTuneRatio := rChillerSystemAnalogInputFineTuneRatio,
    rTargetTempHysteresis := rChillerSystemTempHYSsv,
    rBasedHighTempSV := rChillerSystemTempHALsv,
    rBasedTargetTempSV := rChillerSystemTempSV,
    rBasedTempReadySV := rChillerSystemTempRDYsv,
    rBased1stLimitSV := rChillerSystemTemp1stLimitSv,
    rOverrideTargetTempSV := 0,
    rOverrideTempReadySV := rChillerSystemTempRDYsv,
    rOverride1stLimitSV := rChillerSystemTemp1stLimitSv,
    bHeatingCtrl := FALSE,
    bCoolingCtrl := TRUE,
    bTemperatureOverrideEn := FALSE,
    bManualHeaterOnPB := FALSE,
    bPreparation := bAutoPreparationInt,
    bAutoStart := bAutoStartPB,
    bDeactivatedMode := FALSE,
    iNotReadyAlarmDelayTime := iChillerSystemPreparationTempSv,
    rTemperaturePV => rChillerSystemTempPV,
    bOutputHeaterCooler => bChillerSystemTempOnOff,
    bStatusTempReadyNO => bChillerSystemTempRDY,
    bAlarmHighTempNC => bChillerSystemTempHAL,
    bAlarm1stLimitNO => bChillerSystemTemp1stLimitAlarm,
    bAlarmTemperatureNotReady => bChillerSystemTempPreparationNoRdyAlarm); // fbV2_TempControl

END_PROGRAM

(* stored: Version 1.1.0.1, ProductVersion 3.1.4024.12
   POU TempCtrl: Id {72cf594b-d6a9-4b65-b92e-d6b3ca3b6676}, SpecialFunc None *)
